{attribute 'Tc2GvlVarNames'}
VAR_GLOBAL CONSTANT
	(* System_AFA_Zustand_Status *)
	E_System_AFA_Zustand_Status_Idle_Sperre			: SINT := 0;
	E_System_AFA_Zustand_Status_Betriebsbereit		: SINT := 1;
	E_System_AFA_Zustand_Status_Nachl_Pumpe			: SINT := 2;
	E_System_AFA_Zustand_Status_Vorl_Pumpe			: SINT := 3;
	E_System_AFA_Zustand_Status_Nachl_Regelventil	: SINT := 4;
	E_System_AFA_Zustand_Status_Vorl_Regelventil	: SINT := 5;
	E_System_AFA_Zustand_Status_Betrieb				: SINT := 6;
	E_System_AFA_Zustand_Status_Betrieb_Sperre		: SINT := 7;
	E_System_AFA_Zustand_Status_Stoerung			: SINT := 99;

	(* System_AFA_Zustand_Regelung_Modus *)
	E_System_AFA_Regelung_Modus_Wanddeckentemperierung		: SINT := -4;
	E_System_AFA_Regelung_Modus_Netz						: SINT := -5;

	E_System_AFA_Regelung_Modus_Waermeabsorber_Automatik	: SINT := 1;
	E_System_AFA_Regelung_Modus_Waermeabsorber_DachWaende	: SINT := 2;
	E_System_AFA_Regelung_Modus_Waermeabsorber_Dach			: SINT := 3;
	E_System_AFA_Regelung_Modus_Rueckkuehler_Automatik		: SINT := -1;
	E_System_AFA_Regelung_Modus_Rueckkuehler_DachWaende		: SINT := -2;
	E_System_AFA_Regelung_Modus_Rueckkuehler_Dach			: SINT := -3;

END_VAR

(* stored: Version 1.1.0.1, ProductVersion 3.1.4024.9
   GVL Con_AFA: Id {1052864b-a0cb-456f-9d0e-59aa858262fb} *)
